// Mitsubishi GX Works2 project: PLC_27112022   PLC: FX3G

// global labels: Global1
VAR_GLOBAL
  fruits_input AT M1 : BOOL;
  oranges_input AT D1132 : REAL;
  oranges_tank AT D1100 : REAL;
  clementine_input AT D1134 : REAL;
  clementine_tank AT D1102 : REAL;
  pummels_input AT D1136 : REAL;
  pummels_tank AT D1104 : REAL;
  div_oragne_by_2 AT M2 : BOOL;
END_VAR
VAR_GLOBAL CONSTANT
  two : REAL := 2;
END_VAR
VAR_GLOBAL
  orange_div_two AT D1106 : REAL;
  helper_1 AT M1 : BOOL;
  helper_3 AT M3 : BOOL;
  helper_2 AT M2 : BOOL;
  helper_4 AT M4 : BOOL;
  helper_5 AT M5 : BOOL;
  start_work_day AT X010 : BOOL;
  emergency_button AT X007 : BOOL;
  work_day_started AT Y010 : BOOL;
  start_washing AT X002 : BOOL;
  three_seconds_timer AT TC0 : BOOL;
END_VAR
VAR_GLOBAL CONSTANT
  three_seconds : INT := 30;
END_VAR
VAR_GLOBAL
  three_seconds_timerr AT TS0 : BOOL;
  light_start_washing AT Y005 : BOOL;
END_VAR
VAR_GLOBAL CONSTANT
  const100 : REAL := 100;
END_VAR
VAR_GLOBAL
  sub_orange_tank AT D1108 : REAL;
  washing AT Y010 : BOOL;
END_VAR
VAR_GLOBAL CONSTANT
  const50 : REAL := 50;
END_VAR
VAR_GLOBAL
  washing_clementine_tank AT D1110 : REAL;
END_VAR
VAR_GLOBAL CONSTANT
  const2 : REAL := 2;
END_VAR
VAR_GLOBAL
  half_orange_washing_tank AT D1112 : REAL;
  pummels_washing_tank AT D1114 : REAL;
  start_squeeze AT X001 : BOOL;
  squeeze_started AT Y001 : BOOL;
  helper_6 AT M6 : BOOL;
  squeeze_tank AT D1116 : REAL;
  start_making_juice AT X011 : BOOL;
  counter_two_times AT CC0 : BOOL;
END_VAR
VAR_GLOBAL CONSTANT
  const2word : INT := 2;
END_VAR
VAR_GLOBAL
  counter_two_times_cs AT CS0 : BOOL;
  three_seconds_timer_squeeze AT TC1 : BOOL;
END_VAR
VAR_GLOBAL CONSTANT
  three_seconds_timer_squeeze_tc : INT := 30;
END_VAR
VAR_GLOBAL
  three_seconds_timer_squeeze_ts AT TS1 : BOOL;
  helper_7 AT M7 : BOOL;
  lamp_1_timer AT TC2 : BOOL;
  lamp_1_timer_ts AT TS2 : BOOL;
  lamp_1 AT Y002 : BOOL;
  lamp_2_timer AT TC3 : BOOL;
END_VAR
VAR_GLOBAL CONSTANT
  time_lamp_2 : WORD := 5;
END_VAR
VAR_GLOBAL
  lamp_2_timer_ts AT TS3 : BOOL;
  lamp_2 AT Y003 : BOOL;
  juice_tank AT D1120 : REAL;
  reset_counter AT CC0 : BOOL;
  helper_8 AT M8 : BOOL;
  start_quality_check AT X003 : BOOL;
  saving_analog_input_2 AT D1128 : REAL;
END_VAR
VAR_GLOBAL CONSTANT
  const0 : REAL;
  const1 : REAL := 1;
  const5 : REAL := 5;
END_VAR
VAR_GLOBAL
  helper_9 AT M9 : BOOL;
  five_seconds_timer_tc AT TC4 : BOOL;
END_VAR
VAR_GLOBAL CONSTANT
  five_seconds : INT := 50;
END_VAR
VAR_GLOBAL
  five_seconds_timer_ts AT TS4 : BOOL;
  light_good_quality_check AT Y004 : BOOL;
  storage_tank AT D1130 : REAL;
  counter_for_quality_check AT CC1 : BOOL;
END_VAR
VAR_GLOBAL CONSTANT
  two_times : INT := 2;
END_VAR
VAR_GLOBAL
  counter_for_quality_check_cs AT CS1 : BOOL;
END_VAR
VAR_GLOBAL CONSTANT
  constt400 : REAL := 400;
END_VAR
VAR_GLOBAL
  analog_input_2 AT D8281 : INT;
  helper_10 AT M10 : BOOL;
  helper_11 AT M11 : BOOL;
  helper_12 AT M12 : BOOL;
  helper_13 AT M13 : BOOL;
  end_day_timer AT TC5 : BOOL;
  end_day_timer_ts AT TS5 : BOOL;
  helper_14 AT M14 : BOOL;
  end_day_timer_1 AT TC6 : BOOL;
END_VAR
VAR_GLOBAL CONSTANT
  half : INT := 50;
  half_second : INT := 5;
END_VAR
VAR_GLOBAL
  end_day_timer_1_ts AT TS6 : BOOL;
  end_day_timer_2 AT TC7 : BOOL;
  end_day_timer_2_ts AT TS7 : BOOL;
  yeve AT Y011 : BOOL;
  helper_15 AT M15 : BOOL;
  helper_16 AT M16 : BOOL;
  helper_17 AT M17 : BOOL;
  helper_18 AT M18 : BOOL;
  helper_19 AT M19 : BOOL;
  helper_20 AT M20 : BOOL;
  helper_21 AT M21 : BOOL;
  helper_22 AT M22 : BOOL;
  helper_23 AT M23 : BOOL;
  orange_washing_tank AT D1108 : REAL;
  helper_24 AT M24 : BOOL;
  helper_25 AT M25 : BOOL;
  helper_26 AT M26 : BOOL;
  temp_check AT X005 : BOOL;
  temp AT D1140 : REAL;
END_VAR
VAR_GLOBAL CONSTANT
  const10 : REAL := 10;
END_VAR
VAR_GLOBAL
  helper_27 AT M27 : BOOL;
  helper_28 AT M28 : BOOL;
  temp_timer AT TC8 : BOOL;
  temp_timer_ts AT TS8 : BOOL;
  temp_lamp AT Y006 : BOOL;
  analog_output AT D8282 : INT;
END_VAR
VAR_GLOBAL CONSTANT
  const400word : INT := 400;
  word400 : INT := 400;
END_VAR

// task Task_01 (event TRUE, interval 0, priority 31): POU_01

PROGRAM POU_01
VAR
  lamp : BOOL;
END_VAR
VAR CONSTANT
  time_lamp_1 : WORD := 5;
END_VAR
(* structured ladder/FBD written out as ST: instructions are called as NAME(EN, inputs, outputs); _pN, _eN, _tN stand for wires *)
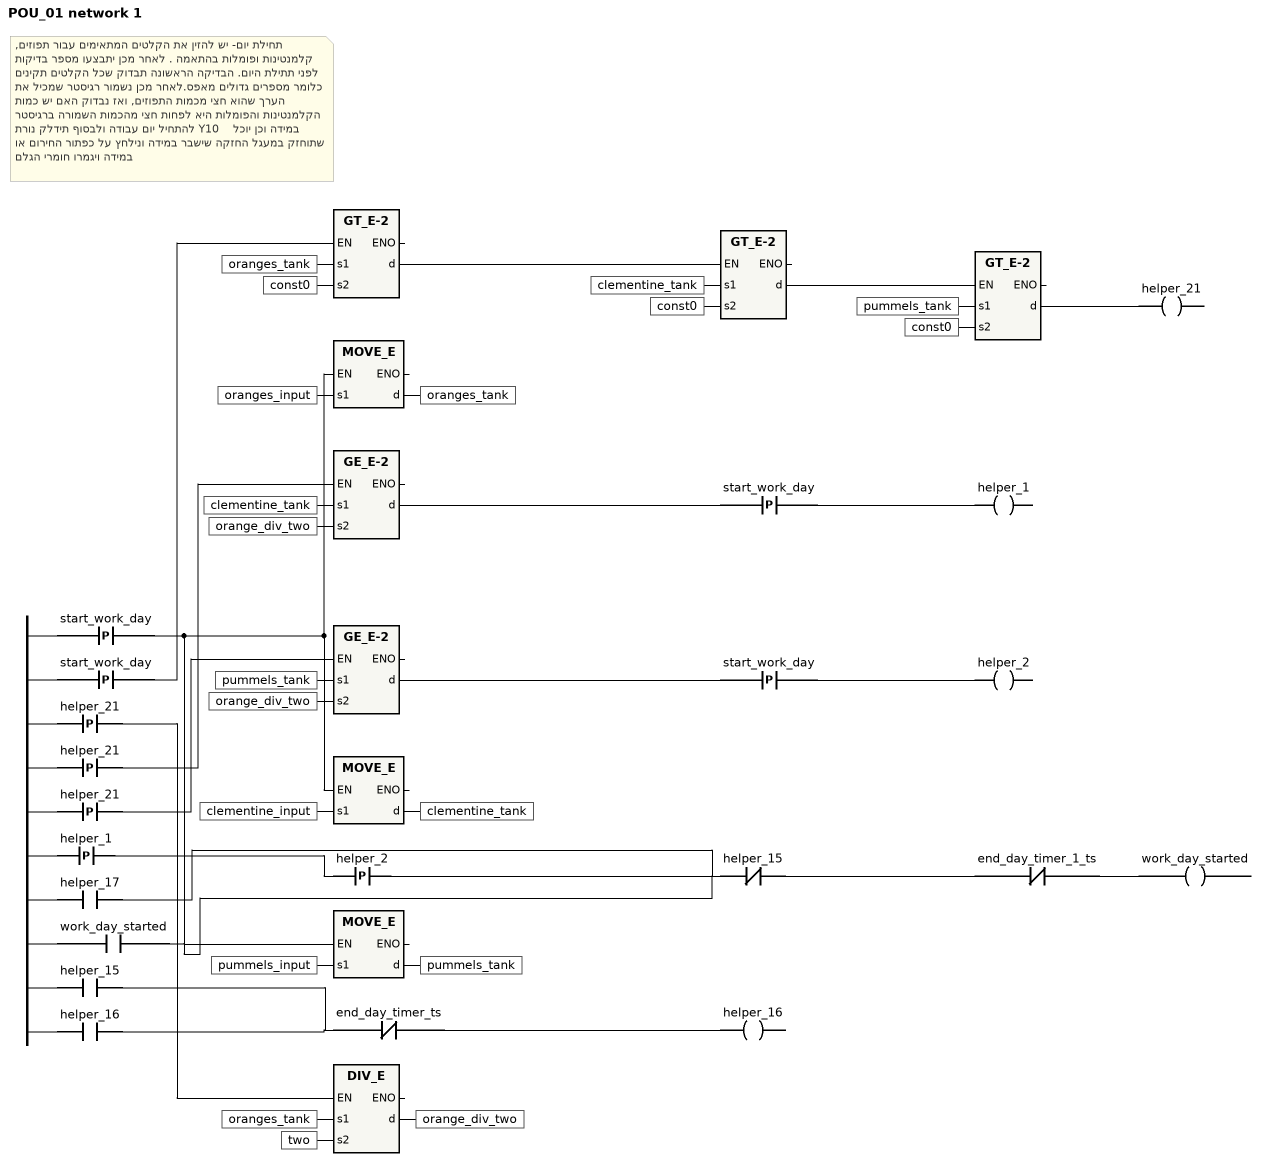
(* network 1 *)
(* תחילת יום- יש להזין את הקלטים המתאימים עבור תפוזים, קלמנטינות ופומלות בהתאמה . לאחר מכן יתבצעו מספר בדיקות לפני תתילת היום. הבדיקה הראשונה תבדוק שכל הקלטים תקינים כלומר מספרים גדולים מאפס.לאחר מכן נשמור רגיסטר שמכיל את הערך שהוא חצי מכמות התפוזים, ואז נבדוק האם יש כמות הקלמנטינות והפומלות היא לפחות חצי מהכמות השמורה ברגיסטר במידה וכן יוכל    Y10 להתחיל יום עבודה ולבסוף תידלק נורת שתוחזק במעגל החזקה שישבר במידה ונילחץ על כפתור החירום או במידה ויגמרו חומרי הגלם *)
_p1 := LDP(TRUE, start_work_day);
MOVE_E(_p1, oranges_input, oranges_tank);
MOVE_E(_p1, clementine_input, clementine_tank);
MOVE_E(_p1, pummels_input, pummels_tank);
GT_E(LDP(TRUE, start_work_day), oranges_tank, const0, _t2);
GT_E(_t2, clementine_tank, const0, _t3);
GT_E(_t3, pummels_tank, const0, _t4);
helper_21 := _t4;
DIV_E(LDP(TRUE, helper_21), oranges_tank, two, orange_div_two);
GE_E(LDP(TRUE, helper_21), clementine_tank, orange_div_two, _t5);
helper_1 := _t5 AND LDP(TRUE, start_work_day);
GE_E(LDP(TRUE, helper_21), pummels_tank, orange_div_two, _t6);
helper_2 := _t6 AND LDP(TRUE, start_work_day);
work_day_started := (((LDP(TRUE, helper_1) AND LDP(TRUE, helper_2)) OR helper_17 OR work_day_started) AND NOT helper_15) AND NOT end_day_timer_1_ts;
helper_16 := (helper_15 OR helper_16) AND NOT end_day_timer_ts;
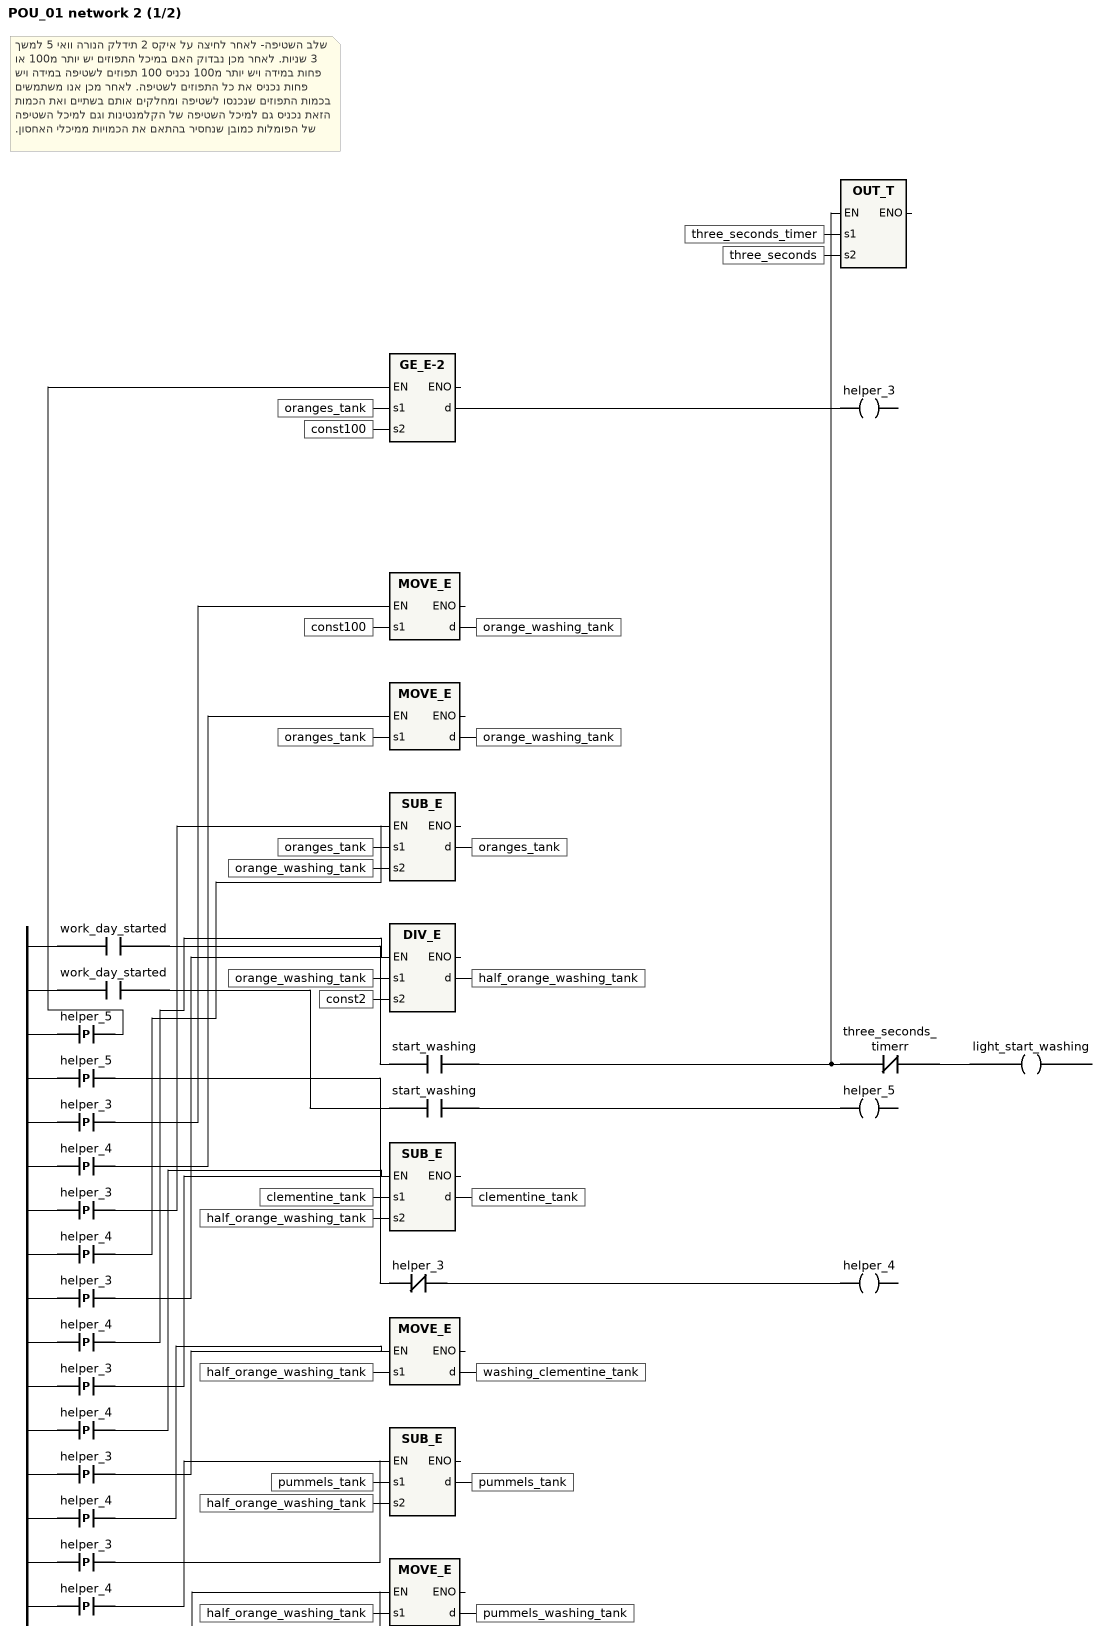
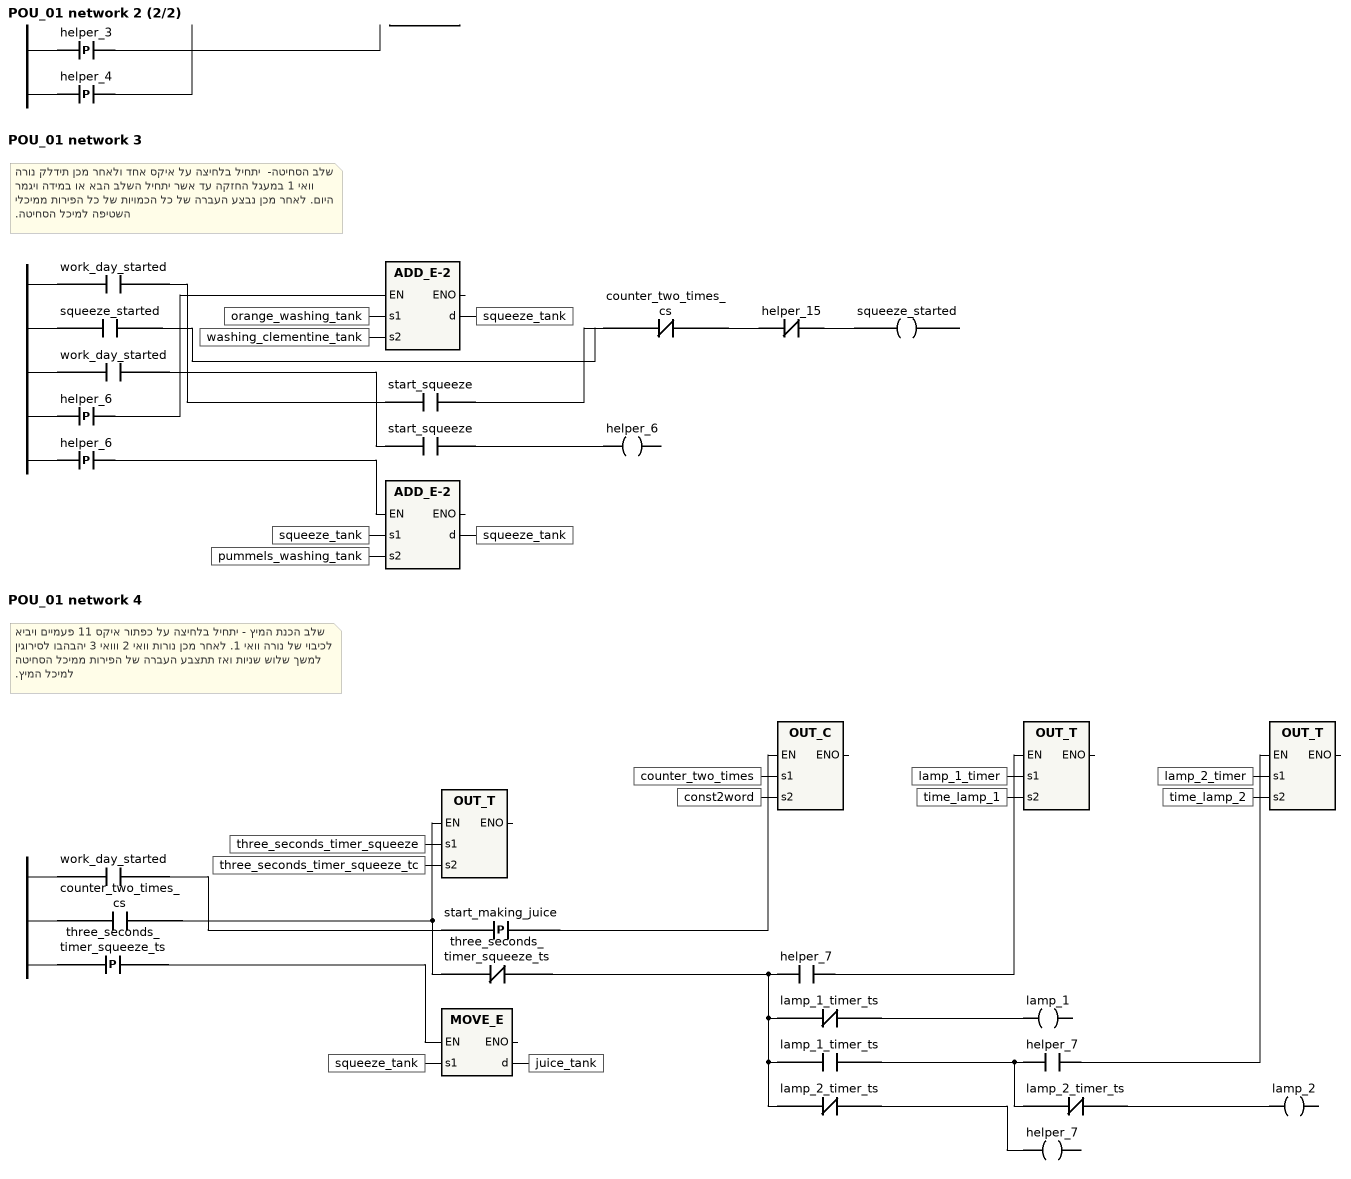
(* network 2 *)
(* שלב השטיפה- לאחר לחיצה על איקס 2 תידלק הנורה וואי 5 למשך 3 שניות. לאחר מכן נבדוק האם במיכל התפוזים יש יותר מ100 או פחות במידה ויש יותר מ100 נכניס 100 תפוזים לשטיפה במידה ויש פחות נכניס את כל התפוזים לשטיפה. לאחר מכן אנו משתמשים בכמות התפוזים שנכנסו לשטיפה ומחלקים אותם בשתיים ואת הכמות הזאת נכניס גם למיכל השטיפה של הקלמנטינות וגם למיכל השטיפה של הפומלות כמובן שנחסיר בהתאם את הכמויות ממיכלי האחסון. *)
_p1 := work_day_started AND start_washing;
OUT_T(_p1, three_seconds_timer, three_seconds);
light_start_washing := _p1 AND NOT three_seconds_timerr;
helper_5 := work_day_started AND start_washing;
GE_E(LDP(TRUE, helper_5), oranges_tank, const100, _t2);
helper_3 := _t2;
helper_4 := LDP(TRUE, helper_5) AND NOT helper_3;
MOVE_E(LDP(TRUE, helper_3), const100, orange_washing_tank);
MOVE_E(LDP(TRUE, helper_4), oranges_tank, orange_washing_tank);
SUB_E(LDP(TRUE, helper_3) OR LDP(TRUE, helper_4), oranges_tank, orange_washing_tank, oranges_tank);
DIV_E(LDP(TRUE, helper_3) OR LDP(TRUE, helper_4), orange_washing_tank, const2, half_orange_washing_tank);
SUB_E(LDP(TRUE, helper_3) OR LDP(TRUE, helper_4), clementine_tank, half_orange_washing_tank, clementine_tank);
MOVE_E(LDP(TRUE, helper_3) OR LDP(TRUE, helper_4), half_orange_washing_tank, washing_clementine_tank);
SUB_E(LDP(TRUE, helper_3) OR LDP(TRUE, helper_4), pummels_tank, half_orange_washing_tank, pummels_tank);
MOVE_E(LDP(TRUE, helper_3) OR LDP(TRUE, helper_4), half_orange_washing_tank, pummels_washing_tank);
(* network 3 *)
(* שלב הסחיטה-  יתחיל בלחיצה על איקס אחד ולאחר מכן תידלק נורה וואי 1 במעגל החזקה עד אשר יתחיל השלב הבא או במידה ויגמר היום. לאחר מכן נבצע העברה של כל הכמויות של כל הפירות ממיכלי השטיפה למיכל הסחיטה. *)
squeeze_started := (((work_day_started AND start_squeeze) OR squeeze_started) AND NOT counter_two_times_cs) AND NOT helper_15;
helper_6 := work_day_started AND start_squeeze;
ADD_E(LDP(TRUE, helper_6), orange_washing_tank, washing_clementine_tank, squeeze_tank);
ADD_E(LDP(TRUE, helper_6), squeeze_tank, pummels_washing_tank, squeeze_tank);
(* network 4 *)
(* שלב הכנת המיץ - יתחיל בלחיצה על כפתור איקס 11 פעמיים ויביא לכיבוי של נורה וואי 1. לאחר מכן נורות וואי 2 ווואי 3 יהבהבו לסירוגין למשך שלוש שניות ואז תתצבע העברה של הפירות ממיכל הסחיטה למיכל המיץ. *)
OUT_C(work_day_started AND LDP(TRUE, start_making_juice), counter_two_times, const2word);
OUT_T(counter_two_times_cs, three_seconds_timer_squeeze, three_seconds_timer_squeeze_tc);
_p1 := counter_two_times_cs AND NOT three_seconds_timer_squeeze_ts;
OUT_T(_p1 AND helper_7, lamp_1_timer, time_lamp_1);
lamp_1 := _p1 AND NOT lamp_1_timer_ts;
_p2 := _p1 AND lamp_1_timer_ts;
OUT_T(_p2 AND helper_7, lamp_2_timer, time_lamp_2);
lamp_2 := _p2 AND NOT lamp_2_timer_ts;
helper_7 := _p1 AND NOT lamp_2_timer_ts;
MOVE_E(LDP(TRUE, three_seconds_timer_squeeze_ts), squeeze_tank, juice_tank);
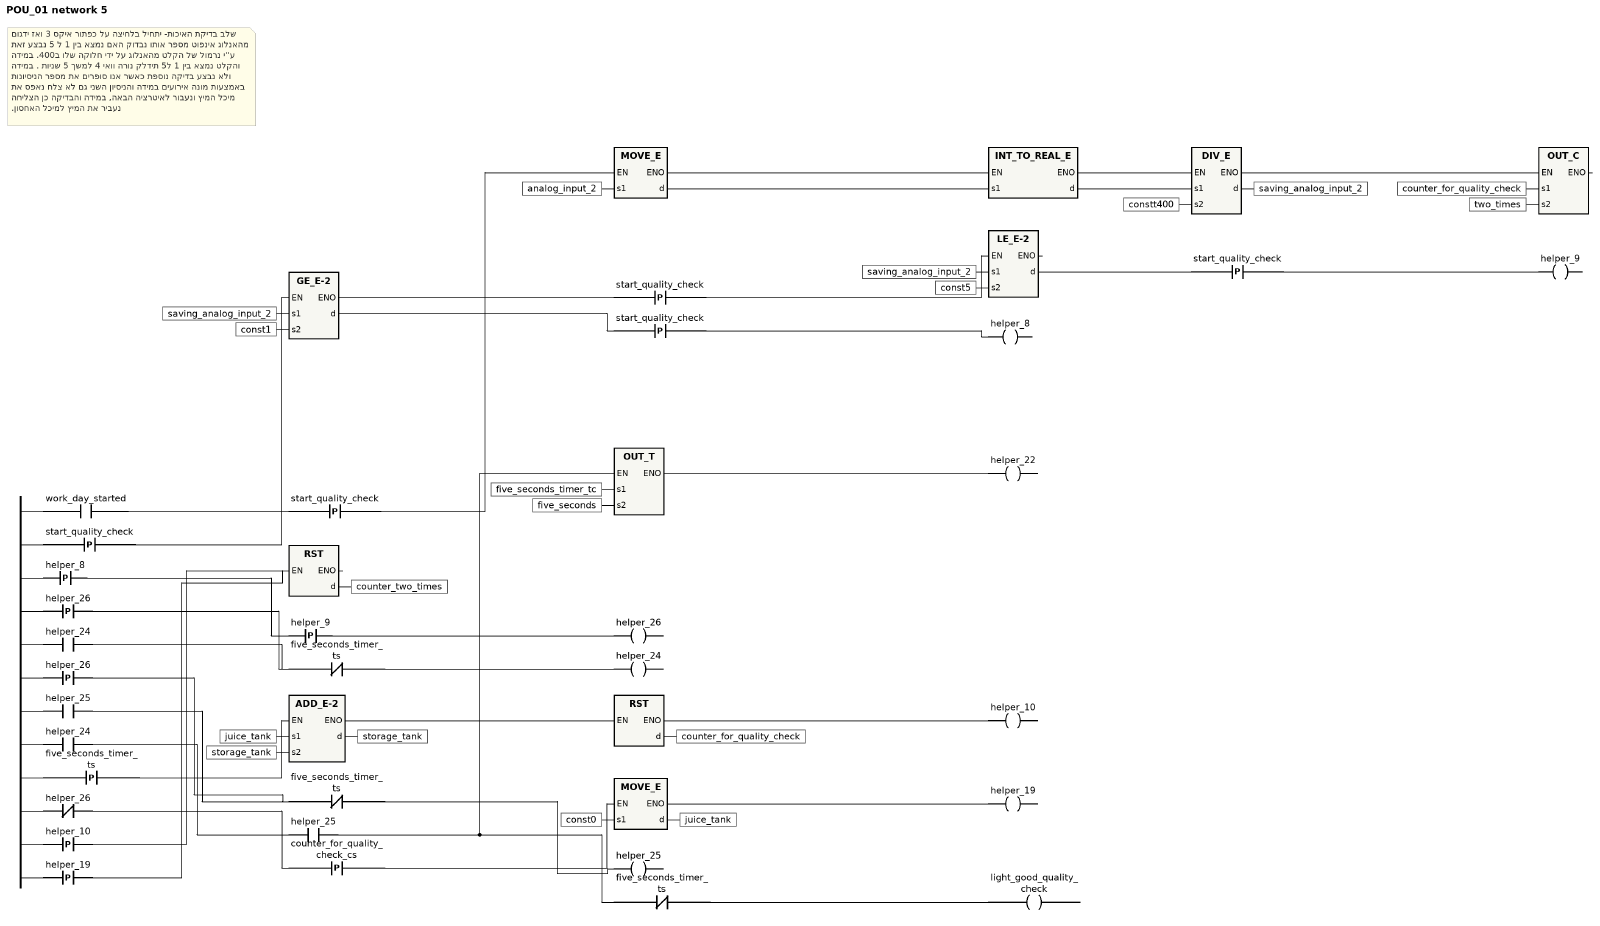
(* network 5 *)
(* שלב בדיקת האיכות- יתחיל בלחיצה על כפתור איקס 3 ואז ידגום מהאנלוג אינפוט מספר אותו נבדוק האם נמצא בין 1 ל 5 נבצע זאת ע''י נרמול של הקלט מהאנלוג על ידי חלוקה שלו ב400. במידה והקלט נמצא בין 1 ל5 תידלק נורה וואי 4 למשך 5 שניות . במידה ולא נבצע בדיקה נוספת כאשר אנו סופרים את מספר הניסיונות באמצעות מונה אירועים במידה והניסיון השני גם לא צלח נאפס את מיכל המיץ ונעבור לאיטרציה הבאה, במידה והבדיקה כן הצליחה נעביר את המיץ למיכל האחסון. *)
_e2 := MOVE_E(work_day_started AND LDP(TRUE, start_quality_check), analog_input_2, _t1);
_e4 := INT_TO_REAL_E(_e2, _t1, _t3);
_e5 := DIV_E(_e4, _t3, constt400, saving_analog_input_2);
OUT_C(_e5, counter_for_quality_check, two_times);
_e7 := GE_E(LDP(TRUE, start_quality_check), saving_analog_input_2, const1, _t6);
LE_E(_e7 AND LDP(TRUE, start_quality_check), saving_analog_input_2, const5, _t8);
helper_8 := _t6 AND LDP(TRUE, start_quality_check);
helper_9 := _t8 AND LDP(TRUE, start_quality_check);
helper_26 := LDP(TRUE, helper_8) AND LDP(TRUE, helper_9);
helper_24 := (LDP(TRUE, helper_26) OR helper_24) AND NOT five_seconds_timer_ts;
helper_25 := (LDP(TRUE, helper_26) OR helper_25) AND NOT five_seconds_timer_ts;
_p9 := helper_24 AND helper_25;
_e10 := OUT_T(_p9, five_seconds_timer_tc, five_seconds);
helper_22 := _e10;
light_good_quality_check := _p9 AND NOT five_seconds_timer_ts;
_e11 := ADD_E(LDP(TRUE, five_seconds_timer_ts), juice_tank, storage_tank, storage_tank);
_e12 := RST(_e11, counter_for_quality_check);
helper_10 := _e12;
_e13 := MOVE_E(NOT helper_26 AND LDP(TRUE, counter_for_quality_check_cs), const0, juice_tank);
helper_19 := _e13;
RST(LDP(TRUE, helper_10) OR LDP(TRUE, helper_19), counter_two_times);
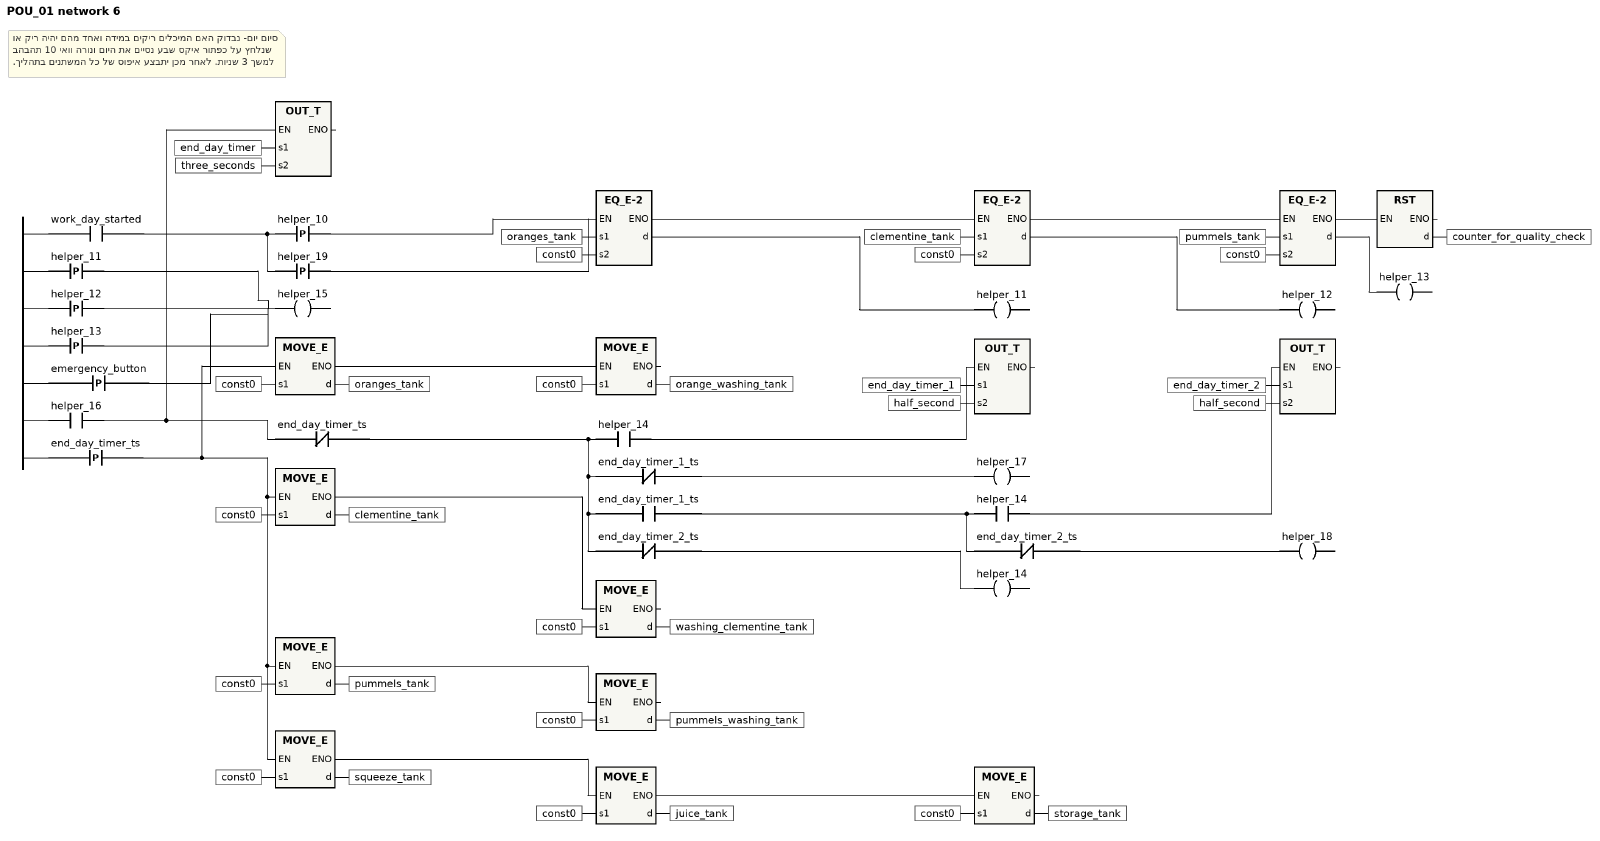
(* network 6 *)
(* סיום יום- נבדוק האם המיכלים ריקים במידה ואחד מהם יהיה ריק או שנלחץ על כפתור איקס שבע נסיים את היום ונורה וואי 10 תהבהב למשך 3 שניות. לאחר מכן יתבצע איפוס של כל המשתנים בתהליך. *)
_e2 := EQ_E((work_day_started AND LDP(TRUE, helper_10)) OR (work_day_started AND LDP(TRUE, helper_19)), oranges_tank, const0, _t1);
_e4 := EQ_E(_e2, clementine_tank, const0, _t3);
_e6 := EQ_E(_e4, pummels_tank, const0, _t5);
RST(_e6, counter_for_quality_check);
helper_11 := _t1;
helper_12 := _t3;
helper_13 := _t5;
helper_15 := LDP(TRUE, helper_11) OR LDP(TRUE, helper_12) OR LDP(TRUE, helper_13) OR LDP(TRUE, emergency_button);
_p7 := helper_16 AND NOT end_day_timer_ts;
OUT_T(_p7 AND helper_14, end_day_timer_1, half_second);
helper_17 := _p7 AND NOT end_day_timer_1_ts;
OUT_T(helper_16, end_day_timer, three_seconds);
_p8 := _p7 AND end_day_timer_1_ts;
OUT_T(_p8 AND helper_14, end_day_timer_2, half_second);
helper_18 := _p8 AND NOT end_day_timer_2_ts;
helper_14 := _p7 AND NOT end_day_timer_2_ts;
_p9 := LDP(TRUE, end_day_timer_ts);
_e10 := MOVE_E(_p9, const0, oranges_tank);
MOVE_E(_e10, const0, orange_washing_tank);
_e11 := MOVE_E(_p9, const0, clementine_tank);
MOVE_E(_e11, const0, washing_clementine_tank);
_e12 := MOVE_E(_p9, const0, pummels_tank);
MOVE_E(_e12, const0, pummels_washing_tank);
_e13 := MOVE_E(_p9, const0, squeeze_tank);
_e14 := MOVE_E(_e13, const0, juice_tank);
MOVE_E(_e14, const0, storage_tank);
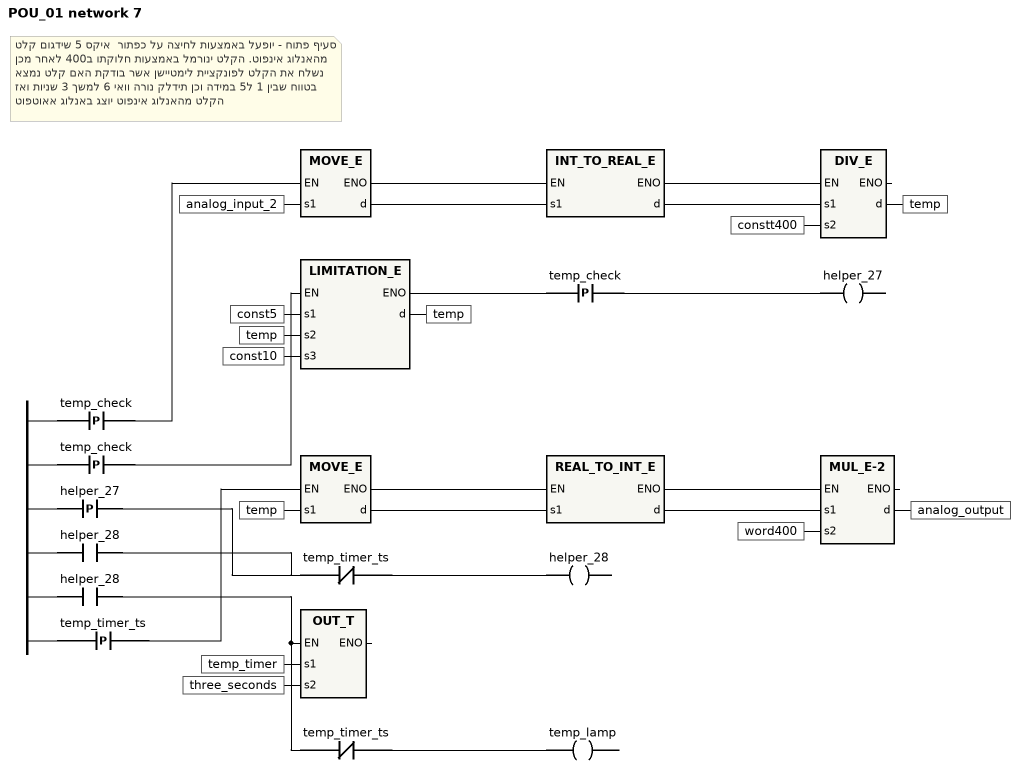
(* network 7 *)
(* סעיף פתוח - יופעל באמצעות לחיצה על כפתור  איקס 5 שידגום קלט מהאנלוג אינפוט. הקלט ינורמל באמצעות חלוקתו ב400 לאחר מכן נשלח את הקלט לפונקציית לימטיישן אשר בודקת האם קלט נמצא בטווח שבין 1 ל5 במידה וכן תידלק נורה וואי 6 למשך 3 שניות ואז הקלט מהאנלוג אינפוט יוצג באנלוג אאוטפוט *)
_e2 := MOVE_E(LDP(TRUE, temp_check), analog_input_2, _t1);
_e4 := INT_TO_REAL_E(_e2, _t1, _t3);
DIV_E(_e4, _t3, constt400, temp);
_e5 := LIMITATION_E(LDP(TRUE, temp_check), const5, temp, const10, temp);
helper_27 := _e5 AND LDP(TRUE, temp_check);
helper_28 := (LDP(TRUE, helper_27) OR helper_28) AND NOT temp_timer_ts;
OUT_T(helper_28, temp_timer, three_seconds);
temp_lamp := helper_28 AND NOT temp_timer_ts;
_e7 := MOVE_E(LDP(TRUE, temp_timer_ts), temp, _t6);
_e9 := REAL_TO_INT_E(_e7, _t6, _t8);
MUL_E(_e9, _t8, word400, analog_output);
END_PROGRAM
